PROGRAM BogieSettings
VAR
	SaveButtonReq : BOOL;
	Saving : bool;		
END_VAR

//set var global via hmi and keep persistient persistient

	WX1Settings();
	WX2Settings();
	WX3Settings();
	WX4Settings();

END_PROGRAM

(* stored: Version 1.1.0.1, ProductVersion 3.1.4024.11
   POU BogieSettings: Id {c604125a-4431-4137-b92c-3fee28a2ef37}, SpecialFunc None *)
